// TwinCAT 3 PLC project Visitor_Pattern
// ProgramVersion: 3.1.4024.0
// libraries:
//   Tc2_Standard, * (Beckhoff Automation GmbH)
//   Tc2_System, * (Beckhoff Automation GmbH)
//   Tc3_Module, * (Beckhoff Automation GmbH)
// project tree:
//   Base Classes/ BaseModuleToBeVisited.TcPOU, ITF_Base.TcIO
//   / PlcTask.TcTTO
//   POUs/ MAIN.TcPOU
//   Visitors/ ITF_Visitor.TcIO, StatusToStringLogVisitor.TcPOU
// (motion and I/O tree: see PLC project simple_factory_pattern)
// real-time tasks:
//   TASK PlcTask: cycle T#10ms, priority 20, ADS port 350
//   TASK PlcTask1: cycle T#10ms, priority 21, ADS port 351
//   TASK PlcTask2: cycle T#10ms, priority 22, ADS port 352
//   TASK PlcTask3: cycle T#10ms, priority 23, ADS port 353
//   TASK PlcTask4: cycle T#10ms, priority 24, ADS port 354
//   TASK PlcTask5: cycle T#10ms, priority 25, ADS port 355
//   TASK PlcTask6: cycle T#10ms, priority 26, ADS port 356
//   TASK PlcTask7: cycle T#10ms, priority 27, ADS port 357
//   TASK PlcTask8: cycle T#10ms, priority 28, ADS port 358
//   TASK PlcTask9: cycle T#10ms, priority 29, ADS port 359

CONFIGURATION Visitor_Pattern
    RESOURCE PLC ON TwinCAT3
        TASK PlcTask(INTERVAL := T#10ms, PRIORITY := 29);
        PROGRAM MAIN WITH PlcTask : MAIN;
    END_RESOURCE
END_CONFIGURATION

// ---- Base Classes/ITF_Base.TcIO
INTERFACE ITF_Base

METHOD GetErrorMessage : String
VAR_INPUT
END_VAR
END_METHOD

METHOD HasError : BOOL
VAR_INPUT
END_VAR
END_METHOD

PROPERTY Name : string
GET
END_GET
END_PROPERTY

END_INTERFACE

// ---- Visitors/ITF_Visitor.TcIO
INTERFACE ITF_Visitor

METHOD VisitBaseObject : BOOL
VAR_INPUT
	BaseObject : ITF_Base;
END_VAR
END_METHOD

END_INTERFACE

// ---- POUs/MAIN.TcPOU
PROGRAM MAIN
VAR
	AxisBaseObject : BaseModuleToBeVisited(MyName := 'axis1');
	Status : T_MaxString;
	statusStringVisitor : StatusToStringLogVisitor(Status);
END_VAR

END_PROGRAM

// ---- Base Classes/BaseModuleToBeVisited.TcPOU
FUNCTION_BLOCK BaseModuleToBeVisited IMPLEMENTS ITF_Base
VAR
	_name : STRING;
	_hasError : BOOL;
	_errorMessage : STRING;
END_VAR

METHOD Accept : BOOL
VAR_INPUT
	Visitor : ITF_Visitor;
END_VAR
Visitor.VisitBaseObject(this^);
END_METHOD

METHOD FB_init : BOOL
VAR_INPUT
	bInitRetains : BOOL; // if TRUE, the retain variables are initialized (warm start / cold start)
	bInCopyCode : BOOL;  // if TRUE, the instance afterwards gets moved into the copy code (online change)
	MyName : STRING;
END_VAR
_name := MyName;
END_METHOD

METHOD GetErrorMessage : STRING
END_METHOD

METHOD HasError : BOOL
HasError := _hasError;
END_METHOD

PROPERTY Name : STRING
GET
Name := _name;
END_GET
END_PROPERTY

END_FUNCTION_BLOCK

// ---- Visitors/StatusToStringLogVisitor.TcPOU
FUNCTION_BLOCK StatusToStringLogVisitor IMPLEMENTS ITF_Visitor
VAR
	StringLog : reference to T_MaxString;
END_VAR

METHOD FB_init : BOOL
VAR_INPUT
	bInitRetains : BOOL; // if TRUE, the retain variables are initialized (warm start / cold start)
	bInCopyCode : BOOL;  // if TRUE, the instance afterwards gets moved into the copy code (online change)
	StringLog : T_MaxString;
END_VAR
END_METHOD

METHOD VisitBaseObject : BOOL
VAR_INPUT
	BaseObject : ITF_Base;
END_VAR
StringLog := CONCAT(StringLog, '[');
StringLog := CONCAT(StringLog, BaseObject.Name);
StringLog := CONCAT(StringLog, ']');

IF BaseObject.HasError() THEN
	StringLog := CONCAT(StringLog, ': Has Error ');
	StringLog := CONCAT(StringLog, BaseObject.GetErrorMessage());
	StringLog := CONCAT(StringLog, '. ');
ELSE
	StringLog := CONCAT(StringLog, ': Has No Error. ');
END_IF
END_METHOD

END_FUNCTION_BLOCK
